// TIA Portal project "20240904" (V15.1)

(* hardware
DEVICE "S7-1200 station_1"  S7-1200 Station
   slot 0: "Rack_0"  S7-1200 Rack  Rack  V1.0
   slot 1: "PLC_1"  CPU 1212C DC/DC/DC  6ES7 212-1AE40-0XB0  V4.2
   slot 2: "DI 16x24VDC/DQ 16xRelay_1"  SM 1223 DI16/DQ16 x relay  6ES7 223-1PL32-0XB0  V2.0
*)

// ===== PLC "PLC_1"  CPU 1212C DC/DC/DC =====

VAR_GLOBAL   // PLC tag table "默认变量表"
   "Tag_1" AT %I8.0 : Bool;
   "Tag_2" AT %M2.0 : Bool;
   "Tag_3" AT %M2.1 : Bool;
   "Tag_4" AT %M2.2 : Bool;
   "Tag_5" AT %Q8.0 : Bool;
   "Tag_6" AT %Q8.1 : Bool;
   "Tag_7" AT %Q8.2 : Bool;
   "Tag_8" AT %Q8.3 : Bool;
   "Tag_9" AT %Q8.4 : Bool;
   "Tag_10" AT %Q8.5 : Bool;
   "Tag_11" AT %Q8.6 : Bool;
   "Tag_12" AT %Q8.7 : Bool;
   "Tag_13" AT %MD100 : Time;
   "Tag_14" AT %M2.3 : Bool;
END_VAR

// folder: System blocks/Program resources

DATA_BLOCK "IEC_Counter_0_DB"   // DB1
{ S7_Optimized_Access := 'TRUE' }
AUTHOR : Simatic
FAMILY : IEC
NAME : CNTR
VERSION : 1.0
// stored: InstanceOfName IEC_COUNTER
"IEC_COUNTER"
BEGIN
END_DATA_BLOCK

DATA_BLOCK "t1"   // DB2
{ S7_Optimized_Access := 'TRUE' }
AUTHOR : Simatic
FAMILY : IEC
NAME : IEC_TMR
VERSION : 1.0
// stored: InstanceOfName IEC_TIMER
"IEC_TIMER"
BEGIN
END_DATA_BLOCK

DATA_BLOCK "t2"   // DB3
{ S7_Optimized_Access := 'TRUE' }
AUTHOR : Simatic
FAMILY : IEC
NAME : IEC_TMR
VERSION : 1.0
// stored: InstanceOfName IEC_TIMER
"IEC_TIMER"
BEGIN
END_DATA_BLOCK

DATA_BLOCK "IEC_Counter_0_DB_1"   // DB4
{ S7_Optimized_Access := 'TRUE' }
AUTHOR : Simatic
FAMILY : IEC
NAME : CNTR
VERSION : 1.0
// stored: InstanceOfName IEC_COUNTER
"IEC_COUNTER"
BEGIN
END_DATA_BLOCK

// folder: (top level)

ORGANIZATION_BLOCK "Main"   // OB1, LAD, ProgramCycle
TITLE = "Main Program Sweep (Cycle)"
{ S7_Optimized_Access := 'TRUE' }
VERSION : 0.1
// congratulation！好好学（ba）习（pia）吧
   VAR_INPUT
      Initial_Call : Bool;   // Initial call of this OB
      Remanence : Bool;   // =True, if remanent data are available
   END_VAR
BEGIN

REGION Network 1
   // 三次按钮
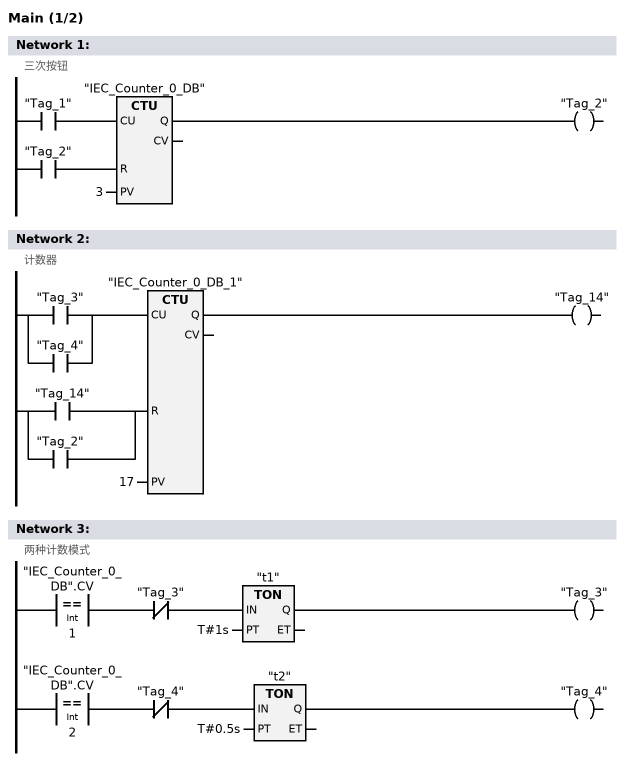
   "IEC_Counter_0_DB".CTU(CU := "Tag_1", R := "Tag_2", PV := 3);
   "Tag_2" := "IEC_Counter_0_DB".Q;
END_REGION

REGION Network 2
   // 计数器
   "IEC_Counter_0_DB_1".CTU(CU := "Tag_3" OR "Tag_4", R := "Tag_14" OR "Tag_2", PV := 17);
   "Tag_14" := "IEC_Counter_0_DB_1".Q;
END_REGION

REGION Network 3
   // 两种计数模式
   "t1".TON(IN := ("IEC_Counter_0_DB".CV = 1) AND NOT "Tag_3", PT := T#1s);
   "Tag_3" := "t1".Q;
   "t2".TON(IN := ("IEC_Counter_0_DB".CV = 2) AND NOT "Tag_4", PT := T#0.5s);
   "Tag_4" := "t2".Q;
END_REGION

REGION Network 4
   // 灯的控制
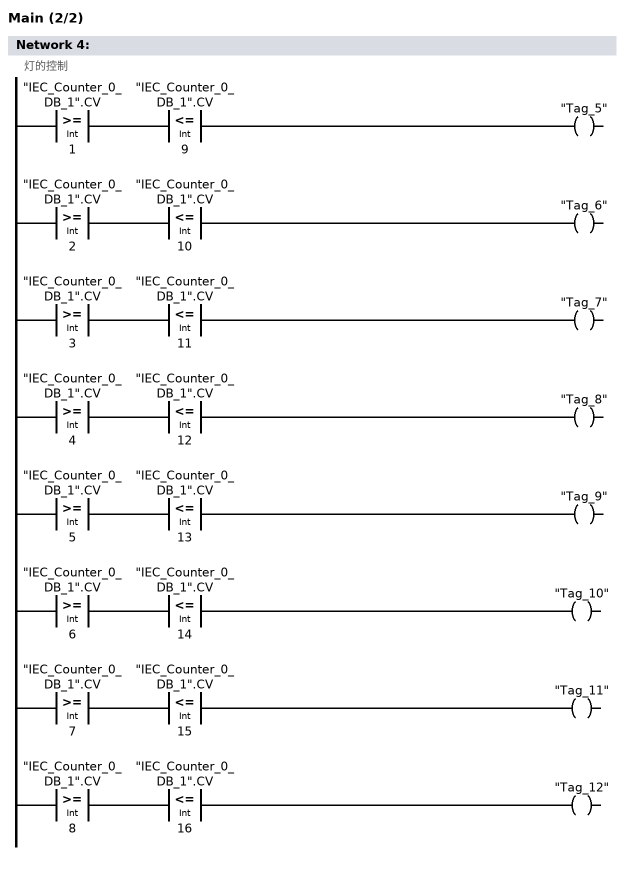
   RUNG wire#powerrail
      { S7_Templates := "SrcType := Int" } GE_Contact(in1 := "IEC_Counter_0_DB_1".CV, in2 := 1)
      { S7_Templates := "SrcType := Int" } LE_Contact(in1 := "IEC_Counter_0_DB_1".CV, in2 := 9)
      Coil( "Tag_5" )
   END_RUNG
   RUNG wire#powerrail
      { S7_Templates := "SrcType := Int" } GE_Contact(in1 := "IEC_Counter_0_DB_1".CV, in2 := 2)
      { S7_Templates := "SrcType := Int" } LE_Contact(in1 := "IEC_Counter_0_DB_1".CV, in2 := 10)
      Coil( "Tag_6" )
   END_RUNG
   RUNG wire#powerrail
      { S7_Templates := "SrcType := Int" } GE_Contact(in1 := "IEC_Counter_0_DB_1".CV, in2 := 3)
      { S7_Templates := "SrcType := Int" } LE_Contact(in1 := "IEC_Counter_0_DB_1".CV, in2 := 11)
      Coil( "Tag_7" )
   END_RUNG
   RUNG wire#powerrail
      { S7_Templates := "SrcType := Int" } GE_Contact(in1 := "IEC_Counter_0_DB_1".CV, in2 := 4)
      { S7_Templates := "SrcType := Int" } LE_Contact(in1 := "IEC_Counter_0_DB_1".CV, in2 := 12)
      Coil( "Tag_8" )
   END_RUNG
   RUNG wire#powerrail
      { S7_Templates := "SrcType := Int" } GE_Contact(in1 := "IEC_Counter_0_DB_1".CV, in2 := 5)
      { S7_Templates := "SrcType := Int" } LE_Contact(in1 := "IEC_Counter_0_DB_1".CV, in2 := 13)
      Coil( "Tag_9" )
   END_RUNG
   RUNG wire#powerrail
      { S7_Templates := "SrcType := Int" } GE_Contact(in1 := "IEC_Counter_0_DB_1".CV, in2 := 6)
      { S7_Templates := "SrcType := Int" } LE_Contact(in1 := "IEC_Counter_0_DB_1".CV, in2 := 14)
      Coil( "Tag_10" )
   END_RUNG
   RUNG wire#powerrail
      { S7_Templates := "SrcType := Int" } GE_Contact(in1 := "IEC_Counter_0_DB_1".CV, in2 := 7)
      { S7_Templates := "SrcType := Int" } LE_Contact(in1 := "IEC_Counter_0_DB_1".CV, in2 := 15)
      Coil( "Tag_11" )
   END_RUNG
   RUNG wire#powerrail
      { S7_Templates := "SrcType := Int" } GE_Contact(in1 := "IEC_Counter_0_DB_1".CV, in2 := 8)
      { S7_Templates := "SrcType := Int" } LE_Contact(in1 := "IEC_Counter_0_DB_1".CV, in2 := 16)
      Coil( "Tag_12" )
   END_RUNG
   // the same network as SCL:
   "Tag_5" := ("IEC_Counter_0_DB_1".CV >= 1) AND ("IEC_Counter_0_DB_1".CV <= 9);
   "Tag_6" := ("IEC_Counter_0_DB_1".CV >= 2) AND ("IEC_Counter_0_DB_1".CV <= 10);
   "Tag_7" := ("IEC_Counter_0_DB_1".CV >= 3) AND ("IEC_Counter_0_DB_1".CV <= 11);
   "Tag_8" := ("IEC_Counter_0_DB_1".CV >= 4) AND ("IEC_Counter_0_DB_1".CV <= 12);
   "Tag_9" := ("IEC_Counter_0_DB_1".CV >= 5) AND ("IEC_Counter_0_DB_1".CV <= 13);
   "Tag_10" := ("IEC_Counter_0_DB_1".CV >= 6) AND ("IEC_Counter_0_DB_1".CV <= 14);
   "Tag_11" := ("IEC_Counter_0_DB_1".CV >= 7) AND ("IEC_Counter_0_DB_1".CV <= 15);
   "Tag_12" := ("IEC_Counter_0_DB_1".CV >= 8) AND ("IEC_Counter_0_DB_1".CV <= 16);
END_REGION
END_ORGANIZATION_BLOCK